PROGRAM MAIN
VAR
	masterAxis : Axis_Ref;
	slaveAxis  : Axis_Ref;
	
	fb_masterStatus : MC_ReadStatus;
	fb_slaveStatus 	: MC_ReadStatus;
	
	fb_masterPower :MC_Power;
	fb_slavePower : MC_Power;
	
	fb_synchronize :MC_GearIn;
	
	fb_moveRelative : MC_MoveRelative;

	
	state		: INT;
	bPower		: BOOL;
	bMove		: BOOL;
	nDistance	: LREAL := 500;
	nVelocity	: LREAL := 50;
END_VAR


CASE state OF
	0: 	//Idle case
	
	fb_masterStatus(
		Axis := masterAxis,
		Enable := TRUE);
		
	fb_slaveStatus(
		Axis := slaveAxis,
		Enable := TRUE);
		
	IF NOT fb_masterStatus.Error AND NOT fb_slaveStatus.Error THEN
		state := 10;
	END_IF
	
	10: 	//Power up motors
	
	IF NOT fb_masterPower.Status THEN
		fb_masterPower.Enable := NOT bPower;
	END_IF
	
	fb_masterPower(
		Axis := masterAxis,
		Enable := bPower,
		Enable_Positive := bPower,
		Enable_Negative := bPower);
		
	fb_slavePower(
		Axis := slaveAxis,
		Enable := bPower,
		Enable_Positive := bPower,
		Enable_Negative := bPower);		
	
	IF fb_masterPower.Status AND fb_slavePower.Status THEN
		state := 20;
	END_IF
	
	20: 	//Synchronize motors
	IF NOT fb_synchronize.InGear THEN
		fb_synchronize.Execute := FALSE;
	END_IF
	
	fb_synchronize(
		Master := masterAxis,
		Slave := slaveAxis,
		Execute := TRUE);
		
	IF fb_synchronize.InGear THEN
		state := 30;
	END_IF

	30: 	//Move relative 500mm at 50mm/s
	
	fb_moveRelative(
		Axis := masterAxis,
		Execute := bMove,
		Distance := nDistance,
		Velocity := nVelocity);
END_CASE

END_PROGRAM

(* stored: Version 1.1.0.1, ProductVersion 3.1.4022.17
   POU MAIN: Id {dffadb6e-f396-4be4-94c2-585b4cb42b02}, SpecialFunc None *)
